(* PLC project KinIn_v3.project, CODESYS CODESYS V3.5 SP19 *)
(* stored: creationDateTime 2025-01-20T16:30:51.4645719, modificationDateTime 2025-01-20T16:30:33.4988497 *)

PROGRAM PLC_PRG
  VAR
    getFwdKinematics_Body : getFwdKinematics_Body;
    Blist : ARRAY[1..6, 1..GVL.nJoints] OF REAL := [0.0, 0.0, -3.20510345E-09, 1.0, 0.0, 0.0, 1.0, -1.0, -3.20510345E-09, 1.0, 1.0, -3.20510345E-09, 3.20510345E-09, 1.02726882E-17, -3.20510345E-09, -0.582899996, -1.1225, 1.147, 3.67625366E-09, -0.882, 2.8498, -8.42878107E-09, -2.98395132E-09, 1.147, -3.6217669E-10, 0.0, -2.6298, 0.216, 0.582899997, -0.113];
    M : ARRAY[1..4, 1..4] OF REAL := [1, 0, 0, 2.8498, 0, 1, 0, 0.5829, 0, 0, 1, -1.1225, 0, 0, 0, 1];
    T_FK : ARRAY[1..4, 1..4] OF REAL;
    T : ARRAY[1..4, 1..4] OF REAL := [0.9206, -0.1413, 0.364, 2309.8, 0.193, 0.9751, -0.1095, 1193.5, -0.3394, 0.171, 0.925, -1424.4, 0, 0, 0, 1.0];  (* ----------IKinematics----- *)
    thetalist_FK : ARRAY[1..GVL.nJoints] OF REAL := [((0 * 3.1415) / 180), ((-10 * 3.1415) / 180), 0, ((10 * 3.1415) / 180), ((10 * 3.1415) / 180)];  (* thetalist0 :ARRAY [1..GVL.nJoints] OF REAL; *)
    thetalist : ARRAY[1..GVL.nJoints] OF REAL;
    eomg : REAL := 0.1;
    ev : REAL := 0.08;
    success : BOOL;
    RndStart : RndStart;  (* -----------for various iterations of IK--------- *)
    i_iteration : DINT;
    nIterationsIK : DINT := 20;
    q_JointOK : BOOL;
    q_IKsuccess : BOOL;
    i : DINT;
    s_IK_message : STRING;
    INV_KINEMATICS : INV_KINEMATICS;  (* ------------------INV_KINEMATICS------------------------ *)
    q_success : BOOL;
  END_VAR

             			 
//Testing Forward kinematics  OK
getFwdKinematics_Body(M:=M , Blist:=Blist , thetalist:=thetalist_FK , T=> T_FK);

//Testing inverse kinematics (uses input from Forward kinematics)
INV_KINEMATICS(
	M:= M, 
	T:= T_FK, 
	eomg:= eomg, 
	ev:= ev, 
	nIterationsIK:= nIterationsIK, 
	Blist:= Blist, 
	thetalist=> thetalist, 
	q_IKsuccess=> q_IKsuccess, 
	s_IK_message=> s_IK_message );

IF q_IKsuccess=TRUE THEN
	q_success:=true;
END_IF


          
END_PROGRAM
